	16#4431: sMsg := '4431 function "External hardware latch activation (encoder)" The activation of the external hardware latch (only available on the KL5101) is initiated explicitly by an ADS command (called from the PLC program of th…';
	16#4432: sMsg := '4432 function "External hardware latch activation (encoder)" If a referencing procedure has previously been initiated and the hardware still signals a valid latch value ("latch valid"), this function must not be ca…';
	16#4433: sMsg := '4433 function "External hardware latch activation (encoder)" If this function has already been initiated and the hardware is still signaling that the external latch value is still valid ("extern latch valid"), a fu…';
	16#4434: sMsg := '4434 monitoring "Encoder function not supported" An encoder function has been activated that is currently not released for use, or which is not even implemented.';
	16#4435: sMsg := '4435 monitoring „Encoder function is already active” An encoder function can not been activated because this functionality is already active.';
	16#4440: sMsg := '4440 initialization "Encoder initialization" Encoder has not been initialized. Although the axis has been created, the rest of the initialization has not been performed (1. Initialization of axis I/O, 2. Initialization o…';
	16#4441: sMsg := '4441 address "Axis address" The encoder does not have an axis, or the axis address has not been initialized.';
	16#4442: sMsg := '4442 address "I/O input structure address" The drive does not have a valid I/O input address in the process image.';
	16#4443: sMsg := '4443 address "I/O output structure address" The encoder does not have a valid I/O output address in the process image.';
	16#4450: sMsg := '4450 monitoring "Encoder counter underflow monitoring" The encoders incremental counter has underflowed.';
	16#4451: sMsg := '4451 monitoring "Encoder counter overflow monitoring" The encoders incremental counter has overflowed.';
	16#4460: sMsg := '4460 monitoring "Software end location minimum (axis start)" With active monitoring of the software end location for a minimum, a start has been made from a position that lies below the software end location minimum.…';
	16#4461: sMsg := '4461 monitoring "Software end location maximum (axis start)" With active monitoring of the software end location for a maximum, a start has been made from a position that lies above the software end location maximum.…';
	16#4462: sMsg := '4462 monitoring "Software end location minimum (positioning process)" With active monitoring of the software end location for a minimum, the actual position has fallen below the software end location minimum. In the …';
	16#4463: sMsg := '4463 monitoring "Software end location maximum (positioning process)" With active monitoring of the software end location for a maximum, the actual position has exceeded the software end location maximum. In the case…';
	16#4464: sMsg := '4464 monitoring „Encoder hardware error” The drive resp. the encoder system reports a hardware error of the encoder. An optimal error code is displayed in the message of the event log.';
	16#4465: sMsg := '4465 monitoring „Position initialization error at system start” At the first initialization of the set position was this for all initialization trials (without over-/under-flow, with underflow and overflow ) out of t…';
	16#4470: sMsg := '4470 monitoring "SSI transformation fault or not finished" The SSI transformation of the FOX 50 module was faulty for some NC-cycles or did not finished respectively.';
	16#44A2: sMsg := '44A2 monitoring "ENCERR_ADDR_CONTROLLER"';
	16#44A3: sMsg := '44A3 monitoring "ENCERR_INVALID_CONTROLLERTYPE"';
	16#4500: sMsg := '4500 parameter "Controller ID not allowed" The value for the controller ID is not allowed, e.g. because it has already been assigned, is less than or equal to zero, or is greater than 255.';
	16#4501: sMsg := '4501 parameter "Controller type not allowed" The value for the controller type is unacceptable because it is not defined. Type 1: P-controller (position) . . . Type 7: High/low speed controller Type 8: Stepper motor…';
	16#4502: sMsg := '4502 parameter "Controller operating mode not allowed" The value for the controller operating mode is not allowed.';
	16#4503: sMsg := '4503 parameter "Weighting of the velocity pre-control not allowed" The value for the percentage weighting of the velocity pre-control is not allowed. The parameter is pre-set to 1.0 (100%) as standard.';
	16#4504: sMsg := '4504 parameter "Following error monitoring (position) not allowed" The value for the activation of the following error monitoring is not allowed.';
	16#4505: sMsg := '4505 parameter "Following error (velocity) not allowed" The value for the activation of the following error monitoring (velocity) is not allowed.';
	16#4506: sMsg := '4506 parameter "Following error window (position) not allowed" The value for the following error window (maximum allowable following error) is not allowed.';
	16#4507: sMsg := '4507 parameter "Following error filter time (position) not allowed" The value for the following error filter time (position) is not allowed.';
	16#4508: sMsg := '4508 parameter "Following error window (velocity) not allowed" The value for the following error window (velocity) is not allowed.';
	16#4509: sMsg := '4509 parameter "Following error filter time (velocity) not allowed" The value for the following error filter time (velocity) is not allowed.';
	16#4510: sMsg := '4510 parameter "Proportional gain Kv or Kp (position controller) not allowed" The value for the proportional gain (Kv factor or Kp factor) is not allowed.';
	16#4511: sMsg := '4511 parameter "Integral-action time Tn (position controller) not allowed" The value for the integral-action time is not allowed (I proportion of the PID T1 controller).';
	16#4512: sMsg := '4512 parameter "Derivative action time Tv (position controller) not allowed" The value for the derivative action time is not allowed (D proportion of the PID T1 controller).';
	16#4513: sMsg := '4513 parameter "Damping time Td (position controller) not allowed" The value for the damping time is not allowed (D proportion of the PID T1 controller). Suggested value: 0.1 * Tv';
	16#4514: sMsg := '4514 function "Activation of the automatic offset compensation not allowed" Activation of the automatic offset compensation is only possible for certain types of controller (with no I component).';
	16#4515: sMsg := '4515 parameter "Additional proportional gain Kv or Kp (position controller) not allowed" The value for the second term of the proportional gain (Kv factor or Kp factor) is not allowed.';
	16#4516: sMsg := '4516 parameter "Reference velocity for additional proportional gain Kv or Kp (position controller) not allowed" The value for the reference velocity percentage data entry, to which the additional proportional gain i…';
	16#4517: sMsg := '4517 parameter "Proportional gain Pa (acceleration proportion) not allowed" The value for the proportional gain (Pa factor) is not allowed.';
	16#4518: sMsg := '4518 parameter "Proportional gain Kv (velocity controller) not allowed" The value for the proportional gain (Kv factor) is not allowed.';
	16#4519: sMsg := '4519 parameter “Reset time Tn (velocity controller) not allowed” The value for the integral-action time is not allowed (I proportion of the PID T1 controller).';
	16#451A: sMsg := '451A address "CONTROLERR_RANGE_ACCJUMPLIMITINGMODE"';
	16#451B: sMsg := '451B address "CONTROLERR_RANGE_ACCJUMPVALUE"';
	16#451C: sMsg := '451C address "CONTROLERR_RANGE_FILTERTIME"';
	16#451D: sMsg := '451D parameter „Dead zone not allowed” The value for the dead zone from the position error or the velocity error (system deviation) is not allowed (only for complex controller with velocity or torque interface).';
	16#4520: sMsg := '4520 parameter ”Rate time Tv (velocity controller) not allowed” The value for the derivative action time is not allowed (D proportion of the PID T1 controller).';
	16#4521: sMsg := '4521 parameter "Damping time Td (velocity controller) not allowed" The value for the damping time is not allowed (D proportion of the PID T1 controller). Suggested value: 0.1 * Tv';
	16#4522: sMsg := '4522 parameter "CONTROLERR_RANGE_IOUTPUTLIMIT"';
	16#4523: sMsg := '4523 parameter "CONTROLERR_RANGE_DOUTPUTLIMIT"';
	16#4524: sMsg := '4524 parameter "CONTROLERR_RANGE_POSIDISABLEWHENMOVING"';
	16#4540: sMsg := '4540 initialization "Controller initialisation" Controller has not been initialised. Although the controller has been created, the rest of the initialisation has not been performed (1. Initialisation of controller, 2. Re…';
	16#4541: sMsg := '4541 address "Axis address" Controller does not know its axis, or the axis address has not been initialised.';
	16#4542: sMsg := '4542 address "Drive address" Controller does not know its drive, or the drive address has not been initialised.';
	16#4550: sMsg := '4550 monitoring "Following error monitoring (position)" With active following error monitoring (position) a following error exceedance has occurred, whose magnitude is greater than the following error window, and who…';
	16#4551: sMsg := '4551 monitoring "Following error monitoring (velocity)" With active following error monitoring (velocity) a velocity following error exceedance has occurred, whose magnitude is greater than the following error window…';
	16#45A0: sMsg := '45A0 monitoring "CONTROLERR_RANGE_AREA_ASIDE"';
	16#45A1: sMsg := '45A1 monitoring "CONTROLERR_RANGE_AREA_BSIDE"';
	16#45A2: sMsg := '45A2 monitoring "CONTROLERR_RANGE_QNENN"';
	16#45A3: sMsg := '45A3 monitoring "CONTROLERR_RANGE_PNENN"';
	16#45A4: sMsg := '45A4 monitoring "CONTROLERR_RANGE_AXISIDPRESP0"';
	16#4600: sMsg := '4600 parameter "Drive ID not allowed" The value for the drive ID is not allowed, e.g. because it has already been assigned, is less than or equal to zero, or is greater than 255.';
	16#4601: sMsg := '4601 parameter "Drive type not allowed" The value for the drive type is unacceptable because it is not defined.';
	16#4602: sMsg := '4602 parameter "Drive operating mode not allowed" The value for the drive operating mode is not allowed. Modus 1: Standard';
	16#4603: sMsg := '4603 parameter "Motor polarity inverted?" The flag for the motor polarity is not allowed. Flag 0: Positive motor polarity Flag 1: Negative motor polarity';
	16#4604: sMsg := '4604 parameter "Drift compensation/velocity offset (DAC offset)" The value for the drift compensation (DAC offset) is not allowed.';
	16#4605: sMsg := '4605 parameter "Reference velocity (velocity pre-control)" The value for the reference velocity (velocity pre-control) is not allowed.';
	16#4606: sMsg := '4606 parameter "Reference output in percent" The value for the reference output in percent is not allowed. The value 1.0 (100 %) usually corresponds to a voltage of 10.0 V.';
	16#4607: sMsg := '4607 parameter "Quadrant compensation factor" The value for the quadrant compensation factor is not allowed.';
	16#4608: sMsg := '4608 parameter "Velocity reference point in percent" The value for the velocity reference point in percent is not allowed. The value 1.0 corresponds to 100 percent.';
	16#4609: sMsg := '4609 parameter "Output reference point in percent" The value for the output reference point in percent is not allowed. The value 1.0 corresponds to 100 percent.';
	16#460A: sMsg := '460A parameter "Minimum or maximum output limit" The values for the minimum and/or maximum output limit is not allowed. This will happen if the range of values is exceeded, the maximum limit is smaller than the mini…';
	16#460B: sMsg := '460B parameter "DRIVEERR_RANGE_MAXINCREMENT"';
	16#460C: sMsg := '460C parameter "DRIVEERR_RANGE_ DRIVECONTROLDWORD"';
	16#460D: sMsg := '460D parameter "DRIVEERR_RANGE_ RESETCYCLECOUNTER"';
	16#460F: sMsg := '460F parameter „Drive torque output scaling is not allowed” The value for the drive torque output scaling (rotary motor) or the force output scaling (linear motor) is not allowed.';
	16#4610: sMsg := '4610 parameter „Drive velocity output scaling is not allowed” The value for the drive velocity output scaling is not allowed.';
	16#4611: sMsg := '4611 parameter "Profi Drive DSC Proportional gain Kpc (position controller) not allowed" The value for the profi drive DSC proportional gain (Kpc factor) is not allowed.';
	16#4612: sMsg := '4612 parameter „Table-ID is invalid” The value for the table-ID is invalid.';
	16#4613: sMsg := '4613 parameter „Table interpolationtype is invalid” The value for the table interpolation-type is invalid.';
	16#4614: sMsg := '4614 parameter „Outputoffset in percent is invalid” The value for the output offset in percent (+/- 1.0) is invalid.';
	16#4615: sMsg := '4615 parameter „Profi Drive DSC scaling factor for calculating Xerr (position controller) is not allowed” The value as profi drive DSC scaling factor for calculating Xerr is invalid.';
	16#4616: sMsg := '4616 parameter „Drive acceleration output scaling is not allowed” The value for the drive acceleration/deceleration output scaling is not allowed.';
	16#4617: sMsg := '4617 parameter „Drive position output scaling is not allowed” The value for the drive position output scaling is not allowed.';
	16#4620: sMsg := '4620 parameter "Bit mask for stepper motor cycle not allowed" A value in the various stepper motor masks for the cycle concerned is not allowed.';
	16#4621: sMsg := '4621 parameter "Bit mask for stepper motor holding current not allowed" The value for the stepper motor holding mask is not allowed.';
	16#4630: sMsg := '4630 monitoring „Overtemperature” The drive resp. terminal detects an overtemperature alarm.';
	16#4631: sMsg := '4631 monitoring „Undervoltage” The drive resp. terminal detects an undervoltage (supply voltage to low).';
	16#4632: sMsg := '4632 monitoring „Wire breakage in phase A” The drive resp. terminal detects a wire breakage in phase A.';
	16#4633: sMsg := '4633 monitoring „Wire breakage in phase B” The drive resp. terminal detects a wire breakage in phase B.';
	16#4634: sMsg := '4634 monitoring „Overcurrent in phase A” The drive resp. terminal detects an overcurrent in phase A.';
	16#4635: sMsg := '4635 monitoring „Overcurrent in Phase B” The drive resp. terminal detects an overcurrent in phase B.';
	16#4636: sMsg := '4636 monitoring „Torque overload (stall situation)” The drive resp. terminal detects a torque overload (stall situation).';
	16#4640: sMsg := '4640 initialization "Drive initialisation" Drive has not been initialised. Although the drive has been created, the rest of the initialisation has not been performed (1. Initialisation of drive I/O, 2. Initialisation of …';
	16#4641: sMsg := '4641 address "Axis address" Drive does not know its axis, or the axis address has not been initialised.';
	16#4642: sMsg := '4642 address "I/O input structure address" The drive does not have a valid I/O input address in the process image.';
	16#4643: sMsg := '4643 address "I/O output structure address" The drive does not have a valid I/O output address in the process image.';
	16#4650: sMsg := '4650 monitoring "Drive not ready for operation" The drive is not ready for operation. The following are possible causes: - the drive is in failure state (hardware fault) - the drive is in the starting-up stage…';
	16#4651: sMsg := '4651 monitoring "Error in cyclic communication with the drive (life counter)"';
	16#4652: sMsg := '4652 monitoring "Not permitted to change the table ID while the axis is enabled"';
	16#4655: sMsg := '4655 monitoring "Invalid IO data for more than n consecutive nc cycles"';
	16#4A00: sMsg := '4A00 parameter "Table ID not allowed" The value for the table ID is not allowed, e.g. because it has already been assigned, is less than or equal to zero, or is greater than 255.';
	16#4A01: sMsg := '4A01 parameter "Table type not allowed" The value for the table type is unacceptable because it is not defined.';
	16#4A02: sMsg := '4A02 parameter "Number of lines in the table not allowed" The value of the number of lines in the table is not allowed, because, for example, it is smaller than two at linear interpolation and smaller than four at s…';
	16#4A03: sMsg := '4A03 parameter "Number of columns in the table is not allowed" The value of the number of columns in the table is not allowed, because, for example, it is less than or equal to zero (depends upon the type of table o…';
	16#4A04: sMsg := '4A04 parameter "Step size (position delta) not allowed" The value for the step size between two lines (position delta) is not allowed, because, for example, it is less than or equal to zero.';
	16#4A05: sMsg := '4A05 parameter "Period not allowed" The value for the period is not allowed, because, for example, it is less than or equal to zero.';
	16#4A06: sMsg := '4A06 parameter "Table is not monotonic" The value for the step size is not allowed, because, for example, it is less than or equal to zero.';
	16#4A07: sMsg := '4A07 initialization „Table sub type is not allowed” The value for the table sub type is not allowed or otherwise the table class (slave type) do not match up to the table main type.';
	16#4A08: sMsg := '4A08 initialization „Table interpolation type is not allowed” The value for the table interpolation type is allowed.';
	16#4A09: sMsg := '4A09 initialization "Incorrect table main type" The table main type is unknown or otherwise the table class (slave type) do not match up to the table main type.';
	16#4A10: sMsg := '4A10 initialization "Table initialisation" Table has not been initialised. Although the table has been created, the rest of the initialisation has not been performed. For instance, the number of lines or columns may be l…';
	16#4A11: sMsg := '4A11 initialization "Not enough memory" Table could not be created, since there is not enough memory.';
	16#4A12: sMsg := '4A12 function "Function not executed, function not available" The function has not been implemented, or cannot be executed, for the present type of table.';
	16#4A13: sMsg := '4A13 function "Line index not allowed" The start line index or the stop line index to be used for read or write access to the table is not allowed. For instance, the line index may be greater than the total number …';
	16#4A14: sMsg := '4A14 function "Column index not allowed" The start column index or the stop column index to be used for read or write access to the table in not allowed. For instance, the column index may be greater than the total…';
	16#4A15: sMsg := '4A15 function "Number of lines not allowed" The number of lines to be read from or written to the table is not allowed. The number of lines must be an integer multiple of the number of elements in a line (n * numbe…';
	16#4A16: sMsg := '4A16 function "Number of columns not allowed" The number of columns to be read from or written to the table is not allowed. The number of columns must be an integer multiple of the number of elements in a column (n…';
	16#4A17: sMsg := '4A17 function "Error in scaling or in range entry" The entries in the table header are inconsistent, e.g. the validity range is empty. If the error is generated during the run time it is a run time error and stops …';
	16#4A18: sMsg := '4A18 function "Multi table slave out of range" The slave master position is outside the table values for the master. The error is a run-time error, and stops the master/slave group.';
	16#4A19: sMsg := '4A19 function "Solo table underflow" The slave master position is outside the table values for the master. The master value of the equidistant table, to be processed linearly, lies under the first table value. The …';
	16#4A1A: sMsg := '4A1A function "Solo table overflow" The slave master position is outside the table values for the master. The master value of the equidistant table, to be processed linearly, lies above the first table value. The e…';
	16#4A1B: sMsg := '4A1B parameter "Incorrect execution mode" The cyclic execution mode can only be "true" or "false".';
	16#4A1C: sMsg := '4A1C parameter "Impermissible parameter" The Fifo parameter is not allowed.';
	16#4A1D: sMsg := '4A1D parameter "Fifo is empty" The Fifo of the external generator is empty. This can signify end of track or a run time error.';
	16#4A1E: sMsg := '4A1E parameter "Fifo is full" The Fifo of the external generator is full. It is the user‘s task to continue to attempt to fill the Fifo with the rejected values.';
	16#4A1F: sMsg := '4A1F parameter „Point-Index of Motion Function invalid” The point index of a Motion Function Point of a Function Table is invalid. First the point index has to be larger than zero and second it has to be numerical c…';
	16#4A20: sMsg := '4A20 initialization „No diagonalisation of matrix” The spline can not be calculated. The master positions are not correct.';
	16#4A21: sMsg := '4A21 initialization „Number of spline points to less” The number of points of a cubic spline has to be greater than two.';
	16#4A22: sMsg := '4A22 initialization „Fifo must not be overwritten” Fifo must not be overwritten since then the active line would be overwritten. It is the task of the user to secure that the active line is not modified.';
	16#4B00: sMsg := '4B00 parameter "Axis has been stopped" The axis has been stopped while the axis moves to target position. The axis could be stopped with a PLC Command via ADS, with the call of AXFNC or with the TwinCAT System Manag…';
	16#4B01: sMsg := '4B01 parameter "Axis cannot be started" The axis cannot be started, because:';
	16#4B02: sMsg := '4B02 parameter "Control mode not allowed" No Target Position Control and no Position Area Control.';
	16#4B03: sMsg := '4B03 parameter "Axis is not moving" Restart position and velocity is only allowed if axis is physically moving.';
	16#4B04: sMsg := '4B04 parameter "Wrong mode for RestartPosAndVelo" Wrong mode.';
	16#4B05: sMsg := '4B05 parameter "Command not allowed"';
	16#4B06: sMsg := '4B06 parameter "Parameter not correct"';
	16#4B07: sMsg := '4B07 parameter "Timeout axis function block"';
	16#4B08: sMsg := '4B08 parameter "Axis in protected mode" Axis is in protected mode (i.e. coupled) and cannot be moved.';
	16#4B09: sMsg := '4B09 parameter "Axis is not ready" Axis is not ready and cannot be moved.';
	16#4B0A: sMsg := '4B0A parameter "Homing error" The Homing of an axis could not be started or was not successful';
	16#4B0B: sMsg := '4B0B parameter "Invalid definition trigger input definition" The definition of the trigger signal used with the function block MC_TouchProbe is invalid. The defined encoder ID, the trigger signal or the trigger sign…';
	16#4B0C: sMsg := '4B0C function "position latch has been deactivated" The function block MC_TouchProbe encountered that a touch probe sequence has been deactivated after the block started this sequence. The reason for instance can b…';
	16#4B0D: sMsg := '4B0D function "Timeout NC status feedback" A function block has successfully executed a command but the NC does not pass the expected feedback in the axis status word.';
	16#4B0E: sMsg := '4B0E function "Supplement not installed" - The function is available as supplement product but not installed on the system.';
	16#4B0F: sMsg := '4B0F function "Timeout Register Access" - The access to a bus terminal register timed out.';
	16#4B10: sMsg := '4B10 function "M-Function request missing" This error occurs if a confirmation of an M-Function is made but the request bit is not set.';
	16#4B11: sMsg := '4B11 parameter "Zero shift index is out of range" The index of the zero shift is invalid';
	16#4B12: sMsg := '4B12 parameter "R parameter index or size is invalid". This error occurs, if the R parameters are written or read and the index or size is out of range';
	16#4B13: sMsg := '4B13 parameter "Index for tool description is invalid"';
	16#4B14: sMsg := '4B14 function "Version of cyclic channel interface does not match to the requested function and function block, resp." This error occurs, if an older TwinCAT Version is used and a new functionality from a newer TcN…';
	16#4B15: sMsg := '4B15 function "Channel is not ready for requested function". The requested function can not be executed due to a wrong state of the channel. This error occurs for instance, if retrace is requested and the axes are …';
	16#4B16: sMsg := '4B16 function "Requested function is not turned on". The requested function requires an explicit activation before it can be executed.';
	16#4B20: sMsg := '4B20 parameter "Cannot append all axes". This error occurs, if you want to append an auxiliary axes to an interpolation group and the function fails. Probably a prior assignment of an auxiliary axes was skipped.';
	16#4B30: sMsg := '4B30 parameter "Pointer invalid". The pointer to a data structure is invalid, e.g. NULL.';
	16#4B31: sMsg := '4B31 parameter "Size of memory invalid". The size parameter is invalid.';
	16#4B32: sMsg := '4B32 parameter "Invalid cam table ID". The cam table ID is out of the range from 1 to 255.';
	16#4B33: sMsg := '4B33 parameter "Invalid point ID". The point ID of a motion function point is lower than 1.';
	16#4B34: sMsg := '4B34 parameter "Invalid number of points ". The number of points to read or write is less than 1.';
	16#4B35: sMsg := '4B35 parameter "Invalid MC table type". The type of a cam table does not match the MC_TableType definition.';
	16#4B36: sMsg := '4B36 parameter "Invalid number of rows". The number of rows of a cam table is less than 1.';
	16#4B37: sMsg := '4B37 parameter "Invalid number of columns". The number of columns of a cam table is invalid.';
	16#4B38: sMsg := '4B38 parameter "Invalid Increment". The increment for an interpolation is invalid, e.g. <= 0.';
	16#4B40: sMsg := '4B40 monitoring "Unsupported Terminal Type". The terminal in use is not supported by this function block.';
	16#4B41: sMsg := '4B41 monitoring "Register Read/Write Error". This error implies to be a validation error.';
	16#4B42: sMsg := '4B42 monitoring "Axis is Enabled". Axis is enabled and is not supposed to be enabled for this operation';
	16#4B43: sMsg := '4B43 parameter "Size of compensation table wrong". The stated table size in bytes is not conform with the real size.';
	16#4B44: sMsg := '4B44 parameter The minimum/ maximum position of the compenstation table is not conform to the position in the table description (ST_CompensationDesc)';
	16#4B45: sMsg := '4B45 parameter "Not implemented". The requested function is not implemented in this combination.';
	16#4B60: sMsg := '4B60 monitoring "Motion command not be activated". A motion command has been started and has been buffered and confirmed by the NC. Nevertheless the command did not become active.';
	16#4B61: sMsg := '4B61 monitoring "Motion command could not be monitored by the PLC". A motion command has been started and has been buffered and confirmed by the NC. The PLC has not been able to monitor the execution of this command……';
	16#4B62: sMsg := '4B62 monitoring "Buffered command finished with error". A buffered command finished with an error. The error number is not available because a new command is already in execution.';
	16#4B63: sMsg := '4B63 monitoring "Buffered command finished without state feedback". A buffered command finished without success or error feedback.';
	16#4B64: sMsg := '4B64 monitoring "  BufferMode  not supported". The  BufferMode  is not supported by the command.';
	16#4B65: sMsg := '4B65 monitoring "Command number is zero". The system administrated command number for buffered commands is zero. ';
	16#4B71: sMsg := '4B71 parameter "Invalid NCI Entry Type". FB_NciFeedTablePreparation is called with an unknown nEntryType';
	16#4B72: sMsg := '4B72 function "NciFeedTable full". The table is full filled and therefore this entry is not accepted.';
	16#4B73: sMsg := '4B73 function internal error';
	16#4B74: sMsg := '4B74 parameter "ST_NciTangentialFollowingDesc: tangential axis is not an auxiliary axis" The entry ST_NciTangentialFollowingDesc contains an tangential axis that is no auxiliary axis.';
	16#4B75: sMsg := '4B75 parameter ST_NciTangentialFollowingDesc: nPathAxis1 and nPathAxis2, resp. are no path axes. So it is not possible to determine the plane.';
	16#4B76: sMsg := '4B76 parameter ST_NciTangentialFollwoingDesc: nPathAxis1 and nPathAxis2 are equal. So it is not possible to determine the plane.';
	16#4B77: sMsg := '4B77 parameter ST_NciGeoCirclePlane: circle is programmed in a wrong manner.';
	16#4B78: sMsg := '4B78 function Internal error in calculation of the tangential following';
	16#4B79: sMsg := '4B79 monitoring Tangential following: With ST_NciTangentialFollowingDesc the monitoring of the deviation angle (E_TfErrorOnCrirical1) is activated and with the actual segment the deviation angle is too big.';
	16#4B7A: sMsg := '4B7A function not implemented';
	16#4B7B: sMsg := '4B7B parameter Tangential Following: The radius of the actual circle segment is too small';
	16#4B7C: sMsg := '4B7C parameter FB_NciFeedTablePreparation: pEntry is NULL';
	16#4B7D: sMsg := '4B7D parameter FB_NciFeedTablePreparation: The specified nEntryType does not match the the structure type';
	16#4B7E: sMsg := '4B7E parameter ST_NciMFuncFast and ST_NciMFuncHsk: The requested m-function is not in between 0..159';
	16#4B7F: sMsg := '4B7F parameter ST_NciDynOvr: The requested value for the dynamic override is not in between 0.01 and 1.0';
	16#4B80: sMsg := '4B80 parameter ST_NciVertexSmoothing: invalid parameter. This error occurs with a negative vertex radius or an unknown vertex smoothing type.';
	16#4B81: sMsg := '4B81 parameter FB_NciFeedTablePrepartion: The requested velocity is not in a valid range';
	16#4B82: sMsg := '4B82 parameter ST_Nci*: invalid parameter';

ELSE
	sMsg := UDINT_TO_STRING(iErrID);
	sMsg := concat(sMsg, ' Unknown Error code');
END_CASE
F_AxErrMsg := sMsg;

END_FUNCTION

// ---- POUs/FB/Various/F_ScaleLREAL.TcPOU
//==================================================================================================
//							Beckhoff Automation Poland
//									30.03.2017
//			Funkcja skalujaca
// 	v1.0	|| TC v 3.1.4020.32		|| - pierwsza wersja
//==================================================================================================
FUNCTION F_ScaleLREAL: LREAL
VAR_INPUT
	lrValue									: LREAL;				// Zmienna skalowana
	lrXmin									: LREAL;				// Dolny zakres zmiennej przeskalowanej
	lrXmax									: LREAL;				// Gorny zakres zmiennej przeskalowanej
	lrYmin									: LREAL;				// Dolny zakres zmiennej skalowanej
	lrYmax									: LREAL;				// Gorny zakres zmiennej skalowanej
	bLimits									: BOOL;					// Ogranicz wyjscie w przedziale lrYmin : lrYmax
END_VAR
VAR
	lrfA									: LREAL;				// Wspolczynnik kierunkowy prostej
	lrfB									: LREAL;				// Wspolczynnik przesuniecia prostej
END_VAR

IF (((lrXmax - lrXmin) < 0.01) AND ((lrXmax - lrXmin) > -0.01)) THEN
	F_ScaleLREAL := lrYmin;
ELSE
	lrfA := (lrYmax - lrYmin) / (lrXmax - lrXmin);
	lrfB := lrYmax - lrfA * lrXmax;
	F_ScaleLREAL := lrfA * lrValue + lrfB;
END_IF;
// LIMITY - opcja
IF bLimits THEN
	IF lrYmin < lrYmax THEN
		F_ScaleLREAL := LIMIT(lrYmin, F_ScaleLREAL, lrYmax);
	ELSE
		F_ScaleLREAL := LIMIT(lrYmax, F_ScaleLREAL, lrYmin);		
	END_IF	
END_IF

END_FUNCTION

// ---- POUs/P00_SensorDiagnostics.TcPOU
PROGRAM P00_SensorDiagnostics
VAR
	fbSensor1: FB_SensorDiag;
END_VAR

ACTION aSensors:
fbSensor1(
	bSensor:= 			P02_BottlePusher.IbBottlePusherBottleBeforeSensor, 
	bReset:=,
	sSensorName:= 		'54B81 - Czujnik przed wbijakiem butelek', 
	bShouldBlinking:= 	P00_PackML.fbPMLAuto.ePMLState = E_PMLState.ePMLState_EXECUTE,						
	tTimeToError:= 		T#60S, 
	bError=>, 
	udiErrorID=>, 
	sErrorStationName=>,
	sErrorDescription=>, 
	sErrorDescription2=>);
	
	
	// 1 przypadek - powinien migać jak jest cykl
END_ACTION

END_PROGRAM

// ---- POUs/P20_ExhaustFan_old.TcPOU
PROGRAM P20_ExhaustFan_old
VAR
		(*****************Wentylator wyciągaowy*******************)
	fbExhaustFan							: FB_MitsubishiInverter;
	fbSensorAcetone							: FB_SensorAcetone;
	fbSensorAirFlow							: FB_SensorFlow;
	
	eExhaustFanState						: E_Station;			
	eExhaustFanRunningState					: E_ConveyorState;	
	fbExhaustFanState						: FB_State;		
	QnExhaustFanVelocitySV					AT %Q*: UDINT; 			(*po kom*)	// Nastawa prędkości transportera
	InExhaustFanVelocityCV 					AT %I*: UDINT;			(*po kom*)
	InExhaustFanSTW 						AT %I*: UINT; 			(*po kom*)	// Statusword transportera wejściowego
	QnExhaustFanCTW 						AT %Q*: UINT;  			(*po kom*)	// Controlword transportera wejsciowego
	InExhaustFanErrorCode 					AT %I*: UINT;			(*po kom*)

	(*** Detekcja acetonu***)
	IbSensorAcetoneDetectionNotError			AT %I* :BOOL;			//Czujnik detekcji acetonu usterka bład
	IbSensorAcetoneDetectionNotLevel2			AT %I* :BOOL;			// Alarm poziomu 2 detekcja acetonu 40%DGW (dolna granica wybuchowści)
	IbSensorAcetoneDetectionNotLevel1			AT %I* :BOOL;			// Alarm poziomu 1 detekcja acetonu 20%DGW (dolna granica wybuchowści)

	QbSensorAcetoneDetectionErrorSafety		AT %Q* :BOOL;			//Czujnik detekcji acetonu usterka bład
	QbSensorAcetoneDetectionLevel2Safety	AT %Q* :BOOL;			// Alarm poziomu 2 detekcja acetonu 40%DGW (dolna granica wybuchowści)
	//IbSensorAcetoneDetectionLevel1Safety	AT %Q* :BOOL;			// Alarm poziomu 1 detekcja acetonu 10%DGW (dolna granica wybuchowści)
	
	(*** Detekcja przepływu powietrza***)
	IbSensorFlowDetectionOK					AT %I* :BOOL;			// Czujnik przepływu powietrza - obencości przepłwu
	IbSensorFlowDetectionError				AT %I* :BOOL;			// Czujnik przepływu powietrza - błąd, alarm
	
	tofbExhaustFanCmdStartDelay: TOF;
	bExTest:BOOL;
END_VAR

aFan();
aSensors();

IF GVL_IO.IbExModeSwitchExMode THEN // SAFETY - PRZEPISANIE
	QbSensorAcetoneDetectionLevel2Safety	:=	IbSensorAcetoneDetectionNotLevel2;
	QbSensorAcetoneDetectionErrorSafety		:=	IbSensorAcetoneDetectionNotError;
ELSE 
	QbSensorAcetoneDetectionLevel2Safety	:=	TRUE;//FALSE;
	QbSensorAcetoneDetectionErrorSafety		:=	TRUE;
END_IF;

IF NOT IbSensorAcetoneDetectionNotLevel1 THEN
	udiExhaustFanVelocitySV:=1500;
ELSE
	udiExhaustFanVelocitySV:=750;
END_IF

VIS.udiExhaustFanVelocityCV:=InExhaustFanVelocityCV; //WIZKA

tofbExhaustFanCmdStartDelay(IN:= bExEnable AND NOT GVL.SensorAcetoneError.bError, PT:=T#3M);
tofbExhaustFanCmdStartDelay.ET;

IF NOT tofbExhaustFanCmdStartDelay.Q THEN
	bExhaustFanEnable		:= FALSE;	
	bExhaustFanCmdStart		:= FALSE;
END_IF

IF bExEnable THEN
	bExhaustFanEnable		:= TRUE;
	bExhaustFanCmdStart		:= TRUE;
END_IF

(*fbExhaustFanState(
	eState													:= eExhaustFanState , 
	bRun													:= bExhaustFanCmdStart,	
	eConveyorRunningState									:= eExhaustFanRunningState , 
	sStateDesc												=> VIS.sExhausFanState,
	iState													=> VIS.iExhausFanState	);*)
	
// Obsługa ostrzeżenia
ExSensorWarning[1].sDescription:=fbSensorAcetone.sWarningDescription;

IF (fbSensorAcetone.bWarning ) AND NOT ExSensorWarning[1].bWarning THEN
	ExSensorWarning[1].bWarning		:=	TRUE;
ELSIF ( NOT fbSensorAcetone.bWarning )AND ExSensorWarning[1].bAcknowledge THEN
	ExSensorWarning[1].bWarning		:=	FALSE;
	ExSensorWarning[1].bAcknowledge	:=	FALSE;
	VIS.uliWarningAcknowledge.24 	:=	FALSE;
ELSIF ExSensorWarning[1].bAcknowledge THEN
	ExSensorWarning[1].bAcknowledge	:=	TRUE;
END_IF

ACTION aFan:
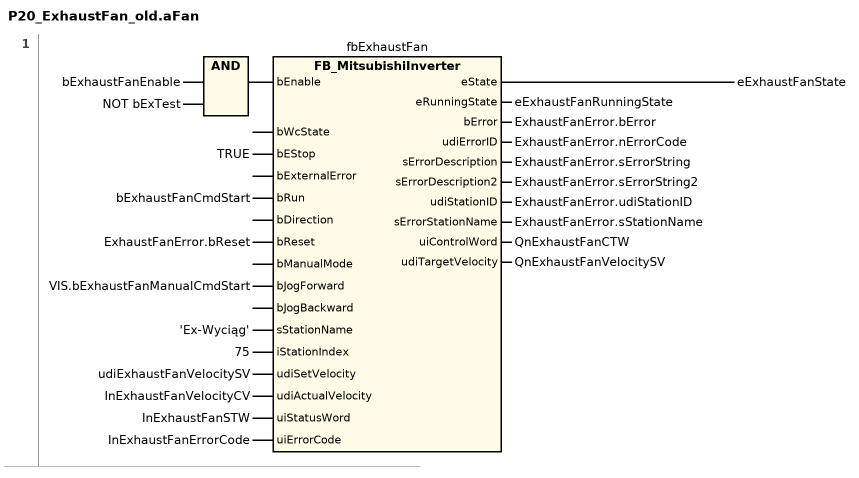
// NETWORK 1
fbExhaustFan(
    bEnable := bExhaustFanEnable AND (NOT bExTest),
    bEStop := TRUE,
    bRun := bExhaustFanCmdStart,
    bReset := ExhaustFanError.bReset,
    bJogForward := VIS.bExhaustFanManualCmdStart,
    sStationName := 'Ex-Wyciąg',
    iStationIndex := 75,
    udiSetVelocity := udiExhaustFanVelocitySV,
    udiActualVelocity := InExhaustFanVelocityCV,
    uiStatusWord := InExhaustFanSTW,
    uiErrorCode := InExhaustFanErrorCode,
    eRunningState => eExhaustFanRunningState,
    bError => ExhaustFanError.bError,
    udiErrorID => ExhaustFanError.nErrorCode,
    sErrorDescription => ExhaustFanError.sErrorString,
    sErrorDescription2 => ExhaustFanError.sErrorString2,
    udiStationID => ExhaustFanError.udiStationID,
    sErrorStationName => ExhaustFanError.sStationName,
    uiControlWord => QnExhaustFanCTW,
    udiTargetVelocity => QnExhaustFanVelocitySV); // FB_MitsubishiInverter
eExhaustFanState := fbExhaustFan.eState;
END_ACTION

ACTION aSensors:
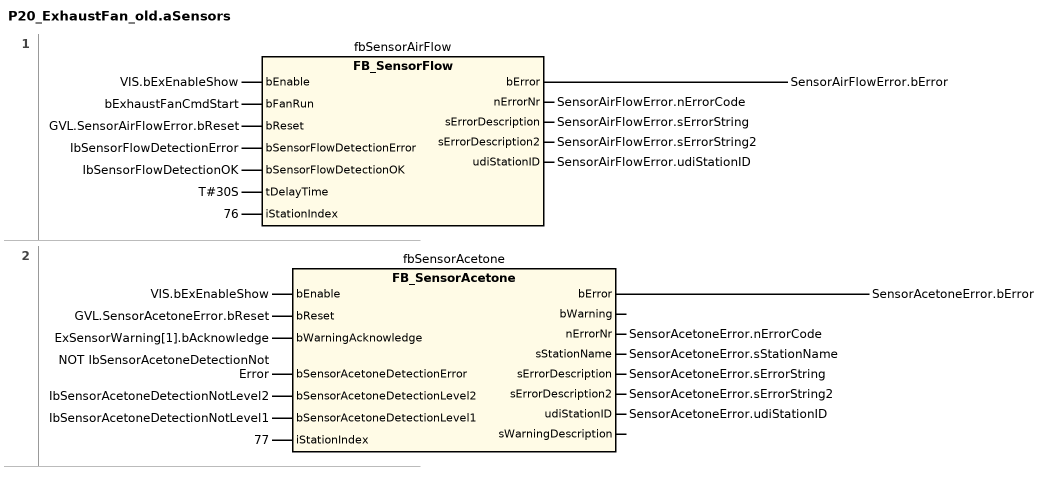
// NETWORK 1
fbSensorAirFlow(
    bEnable := VIS.bExEnableShow,
    bFanRun := bExhaustFanCmdStart,
    bReset := GVL.SensorAirFlowError.bReset,
    bSensorFlowDetectionError := IbSensorFlowDetectionError,
    bSensorFlowDetectionOK := IbSensorFlowDetectionOK,
    tDelayTime := T#30S,
    iStationIndex := 76,
    nErrorNr => SensorAirFlowError.nErrorCode,
    sErrorDescription => SensorAirFlowError.sErrorString,
    sErrorDescription2 => SensorAirFlowError.sErrorString2,
    udiStationID => SensorAirFlowError.udiStationID); // FB_SensorFlow
SensorAirFlowError.bError := fbSensorAirFlow.bError;

// NETWORK 2
fbSensorAcetone(
    bEnable := VIS.bExEnableShow,
    bReset := GVL.SensorAcetoneError.bReset,
    bWarningAcknowledge := ExSensorWarning[1].bAcknowledge,
    bSensorAcetoneDetectionError := NOT IbSensorAcetoneDetectionNotError,
    bSensorAcetoneDetectionLevel2 := IbSensorAcetoneDetectionNotLevel2,
    bSensorAcetoneDetectionLevel1 := IbSensorAcetoneDetectionNotLevel1,
    iStationIndex := 77,
    nErrorNr => SensorAcetoneError.nErrorCode,
    sStationName => SensorAcetoneError.sStationName,
    sErrorDescription => SensorAcetoneError.sErrorString,
    sErrorDescription2 => SensorAcetoneError.sErrorString2,
    udiStationID => SensorAcetoneError.udiStationID); // FB_SensorAcetone
SensorAcetoneError.bError := fbSensorAcetone.bError;
END_ACTION

END_PROGRAM

// ---- POUs/P_WenglorTeach.TcPOU
PROGRAM P_WenglorTeach
VAR
	bTeachModeCapCheck:BOOL;
	bTeachModeCapCorrect:BOOL;
	tofTeachModeCapCheck:TOF;
	tofTeachModeCapCorrect:TOF;
	fbAverageValueCapCheck: FB_Average;
	fbAverageValueCapCorrect: FB_Average;
END_VAR

tofTeachModeCapCheck(IN:=bTeachModeCapCheck,PT:=T#10S);
tofTeachModeCapCorrect(IN:=bTeachModeCapCorrect,PT:=T#10S);
IF tofTeachModeCapCheck.q THEN
	fbAverageValueCapCheck(rValue:=LREAL_TO_REAL(P09_CapPuttedCheck.lrCapPuttedCheckSensorCV), tInterval:= T#5MS, rAverage=>);
END_IF
IF tofTeachModeCapCorrect.q THEN
	fbAverageValueCapCorrect(rValue:=LREAL_TO_REAL(P11_CapCorrectCheck.lrCapCorrectCheckSensorCV), tInterval:= T#5MS, rAverage=>);
END_IF

END_PROGRAM

// ---- POUs/Recipes/NewRecipes/RecipeList/FB_Load.TcPOU
//-----------------------------------------------------------------------------------------------------
//																
//									 	Tkmatik sp z o.o.
//
//	Name					:		FB_Load
//	Author					:		AM
//	Release Date			:		12.01.2022
//	Current ver				:		v 0.1
// 	Last correction 		:		12.01.2022
// 
//	Description				:
//		Special FB for loading structures from BINARY files						
//
//	Requared hardware		:
//
// 	Configuration			:
//
//
//-----------------------------------------------------------------------------------------------------

FUNCTION_BLOCK FB_Load
VAR_INPUT
	sFilePath											:	STRING(255);					//	File path (e.g. 'C:\1.txt')
	pStructAdr											:	PVOID;                          //	Pointer on data struct
	udiStructSize										:	UDINT;                          //	Size of datastruct
	bExecute											:	BOOL;                           //
END_VAR                                                                                     
VAR_OUTPUT                                                                                  
	bBusy												:	BOOL;                           //	FB is Busy
	bDone												:	BOOL;                           //	Load cycle done, DATA actual 
	bError												:	BOOL;                           //	Flag error
	nErrId												:	UDINT;                          //	Error ID
END_VAR                                                                                     
VAR                                                                                         
	fbFileOpen											:	FB_FileOpen;                    //	FB for opening 
	fbFileClose											:	FB_FileClose;                   //	FB for closing
	fbFileRead											:	FB_FileRead;                    //	FB for reading
	hFile												:	UINT;                           //	File hendler
	eMainCase											:	E_FileOpSteps;                  //	Main cycle case value
	rtExecute											:	R_TRIG;                         //	Rtrig for start
END_VAR

ACT_FBs();
ACT_Main();

ACTION ACT_FBs:
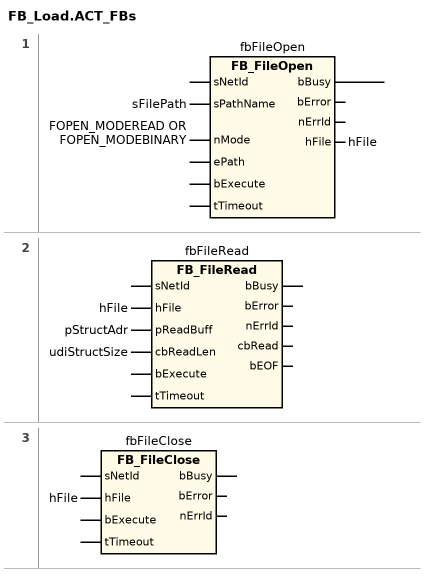
// NETWORK 1
fbFileOpen(sPathName := sFilePath, nMode := FOPEN_MODEREAD OR FOPEN_MODEBINARY, hFile => hFile); // FB_FileOpen

// NETWORK 2
fbFileRead(hFile := hFile, pReadBuff := pStructAdr, cbReadLen := udiStructSize); // FB_FileRead

// NETWORK 3
fbFileClose(hFile := hFile); // FB_FileClose
END_ACTION

ACTION ACT_Main:
rtExecute(CLK:=bExecute);
IF (NOT bExecute) THEN
	bDone												:=	FALSE;
END_IF

CASE eMainCase OF
	E_FileOpSteps.eNop:
		fbFileClose.bExecute							:=	FALSE;
		fbFileOpen.bExecute								:=	FALSE;
		fbFileRead.bExecute								:=	FALSE;
		bBusy											:=	FALSE;
		
		IF (rtExecute.Q) THEN
			bError										:=	FALSE;
			nErrId										:=	0;
			eMainCase									:=	E_FileOpSteps.eStartOpen;
			bBusy										:=	TRUE;
		END_IF
		
	E_FileOpSteps.eStartOpen:
		fbFileOpen.bExecute								:=	TRUE;
		eMainCase										:=	E_FileOpSteps.eWaitOpen;

	E_FileOpSteps.eWaitOpen:
		IF (fbFileOpen.bError) THEN
			bError										:=	TRUE;
			nErrId										:=	10;
			eMainCase									:=	E_FileOpSteps.eNop;
		ELSIF (NOT fbFileOpen.bBusy) THEN
			fbFileOpen.bExecute							:=	FALSE;
			eMainCase									:=	E_FileOpSteps.eStartOper;
		END_IF
		
	E_FileOpSteps.eStartOper:
		fbFileRead.bExecute								:=	TRUE;
		eMainCase										:=	E_FileOpSteps.eWaitOper;
		
	E_FileOpSteps.eWaitOper:
		IF (fbFileRead.bError) THEN
			bError										:=	TRUE;
			nErrId										:=	20;
			eMainCase									:=	E_FileOpSteps.eNop;
		ELSIF (NOT fbFileRead.bBusy) THEN
			fbFileRead.bExecute							:=	FALSE;
			eMainCase									:=	E_FileOpSteps.eStartClose;
		END_IF
		
	E_FileOpSteps.eStartClose:
		fbFileClose.bExecute							:=	TRUE;
		eMainCase										:=	E_FileOpSteps.eWaitClose;
	
	E_FileOpSteps.eWaitClose:
		IF (fbFileClose.bError) THEN
			bError										:=	TRUE;
			nErrId										:=	30;
			eMainCase									:=	E_FileOpSteps.eNop;
		ELSIF (NOT fbFileClose.bBusy) THEN
			fbFileClose.bExecute						:=	FALSE;
			bDone										:=	TRUE;
			eMainCase									:=	E_FileOpSteps.eNop;
		END_IF	
		
END_CASE
END_ACTION

END_FUNCTION_BLOCK

// ---- POUs/Recipes/NewRecipes/RecipeList/FB_Save.TcPOU
//-----------------------------------------------------------------------------------------------------
//																
//									 	Tkmatik sp z o.o.
//
//	Name					:		FB_Save
//	Author					:		AM
//	Release Date			:		12.01.2022
//	Current ver				:		v 0.1
// 	Last correction 		:		12.01.2022
// 
//	Description				:
//		Special FB for saving structures to BINARY files						
//
//	Requared hardware		:
//
// 	Configuration			:
//
//
//-----------------------------------------------------------------------------------------------------

FUNCTION_BLOCK FB_Save
VAR_INPUT
	sFilePath											:	STRING(255);					//	File path (e.g. 'C:\1.txt'
	pStructAdr											:	PVOID;                          //	Pointer on data struct
	udiStructSize										:	UDINT;                          //	Size of datastruct
	bExecute											:	BOOL;                           //
END_VAR                                                                                     
VAR_OUTPUT                                                                                  
	bBusy												:	BOOL;                           //	FB is Busy
	bDone												:	BOOL;                           //	Load cycle done, DATA actual 
	bError												:	BOOL;                           //	Flag error
	nErrId												:	UDINT;                          //	Error ID
END_VAR                                                                                     
VAR                                                                                         
	fbFileOpen											:	FB_FileOpen;                    //	FB for opening 
	fbFileClose											:	FB_FileClose;                   //	FB for closing
	fbFileWrite											:	FB_FileWrite;                   //	FB for saving
	hFile												:	UINT;                           //	File hendler
	eMainCase											:	E_FileOpSteps;                  //	Main cycle case value
	rtExecute											:	R_TRIG;                         //	Rtrig for start
END_VAR

ACT_FBs();
ACT_Main();

ACTION ACT_FBs:
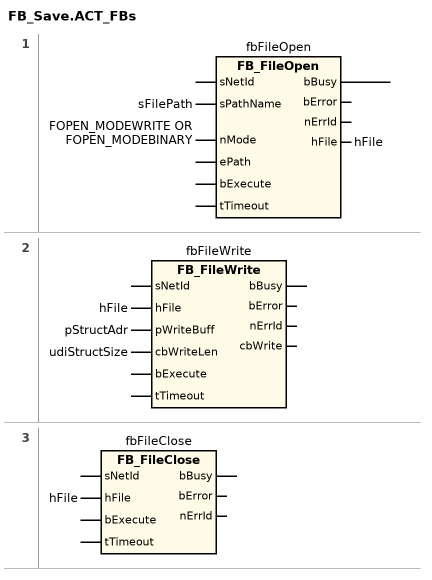
// NETWORK 1
fbFileOpen(sPathName := sFilePath, nMode := FOPEN_MODEWRITE OR FOPEN_MODEBINARY, hFile => hFile); // FB_FileOpen

// NETWORK 2
fbFileWrite(hFile := hFile, pWriteBuff := pStructAdr, cbWriteLen := udiStructSize); // FB_FileWrite

// NETWORK 3
fbFileClose(hFile := hFile); // FB_FileClose
END_ACTION

ACTION ACT_Main:
rtExecute(CLK:=bExecute);
IF (NOT bExecute) THEN
	bDone												:=	FALSE;
END_IF

CASE eMainCase OF
	E_FileOpSteps.eNop:
		fbFileClose.bExecute							:=	FALSE;
		fbFileOpen.bExecute								:=	FALSE;
		fbFileWrite.bExecute							:=	FALSE;
		bBusy											:=	FALSE;
		
		IF (rtExecute.Q) THEN
			bError										:=	FALSE;
			nErrId										:=	0;
			eMainCase									:=	E_FileOpSteps.eStartOpen;
			bBusy										:=	TRUE;
		END_IF
		
	E_FileOpSteps.eStartOpen:
		fbFileOpen.bExecute								:=	TRUE;
		eMainCase										:=	E_FileOpSteps.eWaitOpen;

	E_FileOpSteps.eWaitOpen:
		IF (fbFileOpen.bError) THEN
			bError										:=	TRUE;
			nErrId										:=	10;
			eMainCase									:=	E_FileOpSteps.eNop;
		END_IF
		IF (NOT fbFileOpen.bBusy) THEN
			fbFileOpen.bExecute							:=	FALSE;
			eMainCase									:=	E_FileOpSteps.eStartOper;
		END_IF
		
	E_FileOpSteps.eStartOper:
		fbFileWrite.bExecute							:=	TRUE;
		eMainCase										:=	E_FileOpSteps.eWaitOper;
		
	E_FileOpSteps.eWaitOper:
		IF (fbFileWrite.bError) THEN
			bError										:=	TRUE;
			nErrId										:=	20;
			eMainCase									:=	E_FileOpSteps.eNop;
		END_IF
		IF (NOT fbFileWrite.bBusy) THEN
			fbFileWrite.bExecute						:=	FALSE;
			eMainCase									:=	E_FileOpSteps.eStartClose;
		END_IF
		
	E_FileOpSteps.eStartClose:
		fbFileClose.bExecute							:=	TRUE;
		eMainCase										:=	E_FileOpSteps.eWaitClose;
	
	E_FileOpSteps.eWaitClose:
		IF (fbFileClose.bError) THEN
			bError										:=	TRUE;
			nErrId										:=	30;
			eMainCase									:=	E_FileOpSteps.eNop;
		END_IF
		IF (NOT fbFileClose.bBusy) THEN
			fbFileClose.bExecute						:=	FALSE;
			bDone										:=	TRUE;
			eMainCase									:=	E_FileOpSteps.eNop;
		END_IF	
		
END_CASE
END_ACTION

END_FUNCTION_BLOCK

// ---- GlobalTextList.TcGTLO
TEXTLIST GlobalTextList
  348 = ' '
  627 = '%5.1f'
  520 = '%s'
  835 = 'bFirstPositioningDone'
  928 = 'Chwytak'
  820 = 'Chwytak Homing'
  630 = 'Chwytak pozycja'
  720 = 'Chwytak RUN'
  460 = 'Chwytak stan'
  645 = 'Czas przytrz. %d ms'
  526 = 'Dodatkowy ruch chwytakiem przed zakręceniem  (w poz. doc.)'
  661 = 'Ilość obrotów %5.1f'
  911 = 'Krotność gwintu %5.1f'
  560 = 'kąt szukania gwintu %5.1f'
  899 = 'Kąt szukania gwintu %5.1f'
  644 = 'Manual Mode'
  261 = 'Moment %5.1f'
  402 = 'Obrót %5.1f'
  378 = 'Obrót do tyłu w pozycji dociskania (w trakcie przejazdu do poz. doc.)'
  671 = 'Obrót z pozycji docisku do zakręcania'
  889 = 'Otwarty chwytak przy szukaniu gwintu\t'
  994 = 'Poz. chwyt. butelki %5.1f mm'
  588 = 'Poz. chwyt. butelki %d mm'
  137 = 'Poz. docisku %5.1f mm'
  291 = 'Poz. gotowości %5.1f mm'
  28 = 'Poz. zakręcania %5.1f mm'
  425 = 'Prędkość %5.1f'
  67 = 'ScrewerRun'
  493 = 'Siła chwyt. butelki %5.1f kg'
  252 = 'Siła chwyt. nasadki %5.1f kg'
  113 = 'Siła chwytania nasadki %5.1f kg'
  564 = 'Siła docisku %5.1f kg'
  549 = 'Siła docisku%5.1f kg'
  424 = 'Skok gwintu %5.1f'
  490 = 'Szukanie gwintu w pozycji dociskania\t'
  448 = 'Szukanie gwintu w pozycji zakręcania'
  580 = 'Szukanie gwintu z czujnikiem wysokości'
  430 = 'Tryb momentowy'
  304 = 'Typ głowicy %d'
  841 = 'Typ zakręcania %d'
  505 = 'Wysokość %5.1f'
  844 = 'Wysokość %5.2F mm'
  393 = 'Wysokość %d'
  787 = 'Zak. Homing'
  301 = 'Zak. Reset'
  888 = 'Zakręcarka'
  665 = 'Zakręcarka Manual DOWN'
  333 = 'Zakręcarka Manual UP'
  712 = 'Zakręcarka stan'
END_TEXTLIST
